// TIA Portal V20 export
TYPE "OEM_Data"
// stored: Namespace CITI_Logic
   STRUCT
      Assistance_Call : Array[1..8] of Bool;   // Assistance Call 1 to 8
      Assistance_CallAck : Array[1..8] of Bool;   // Assistance Call Ack 1 to 8
      OUT_TL_Call : Bool;   // Team Lead Call Out
      PMC : "CITI_Logic.PMC_Input_Data";   // PMC Data
      CITI_OneShot { S7_SetPoint := 'True'} : Array[1..32] of Bool;   // CITI One Shot Array
      System_Byte : Byte;   // System Byte
      FirstScan : Bool;   // First Scan
      Always_OFF : Bool;   // Always OFF
      Always_ON : Bool;   // Always ON
      DiagStatusUpdate : Bool;   // Diag Status Update
      Clock_Byte : Byte;   // Clock Byte
      ClockMemByte_Example : Byte;   // Clock Memory Byte Example
      Null_String : String;   // Null String
      TO_COMPLETE : Bool;   // TO COMPLETE
      TO_COMPLETE_INT : Int;   // TO COMPLETE INTEGER
      RESERVED : Byte;   // RESERVED
      MachineFaultedLevel1 : Bool;   // Machine Faulted Level 1
      MachineFaultedLevel2 : Bool;   // Machine Faulted Level 2
      FaultString : String[200];   // Fault String
      Empty_Pallet : Bool;   // Empty Pallet
      OUT_ShiftNumber : Byte;   // OUT Shift Number
      OUT_Flasher : Bool;   // OUT Flasher
      LampCheck : Bool;   // Lamp Check
      Red_Light : Bool;   // Red Stack Light
      Green_Light : Bool;   // Green Stack Light
      Blue_Light : Bool;   // Blue Stack Light
      Yellow_Light : Bool;   // Yellow Stack Light
      No_Maps_Have_Fault_Delay : IEC_TIMER;   // No Maps Have Fault Delay
      IN_Fault_String_Null { S7_SetPoint := 'True'} : Bool;   // IN Fault String Null
      Fault_String_is_Null : Bool;   // Fault String is Null
      FlexNet : "CITI_Logic.FlexNet_Data";   // FlexNet
      FlexNet_Response_Fault_Count { S7_SetPoint := 'True'} : Int;   // FlexNet Response Fault Count
      FlexNet_No_Response_Fault : Bool;   // FlexNet No Response Fault
      FlexNet_No_Response_Warning : Bool;   // FlexNet No Response Warning
      FlexNet_Transaction_Retry_Occurred : Bool;   // FlexNet Transaction Retry Occurred
      FlexNet_DataReceivedByHost : Bool;   // FlexNet Data Received By Host Delayed
      FlexNet_Response_FLT_Time : S5Time;   // FlexNet Response Fault Time
   END_STRUCT;
END_TYPE
